// TIA Portal V18 export
// export: Created 2026-06-14T16:12:11.9430968Z, ExportSetting WithDefaults, DisplayName Totally Integrated Automation Portal, DisplayVersion V18 Update 5, DisplayName TIA Portal Openness, DisplayVersion V18 Update 5, DisplayName TIA Portal Version Control Interface, DisplayVersion V18, DisplayName SINAMICS Startdrive Advanced, DisplayVersion V18 SP2 Update 1, DisplayName SINAMICS Startdrive G110M, G120, G120C, G120D, G120P, G115D, DisplayVersion V18 SP2 Update 1, DisplayName SINAMICS Startdrive G130, G150, S120, S150, SINAMICS MV, S210, G220, S200, DisplayVersion V18 SP2 Update 1, DisplayName STEP 7 Professional, DisplayVersion V18 Update 5, DisplayName STEP 7 Safety, DisplayVersion V18, DisplayName WinCC Advanced / Unified PC, DisplayVersion V18 Update 5
FUNCTION "TEMPLATE--v1.0--06_Feedback Error" : Void   // FC7, F_LAD
TITLE = group / bypass contactor feedback errors by I/O Node
{ S7_Optimized_Access := 'TRUE' }
VERSION : 0.1
// v1.0 First Emission
// stored: AutoNumber true, IsIECCheckEnabled false, UDAEnableTagReadback false
BEGIN

REGION Network 1: !!NetworkComment$$
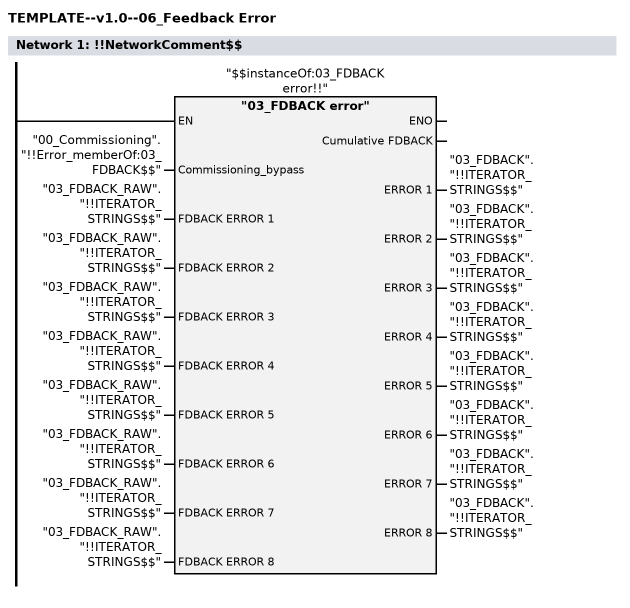
   RUNG wire#powerrail
      "$$instanceOf:03_FDBACK error!!"(Commissioning_bypass := "00_Commissioning"."!!Error_memberOf:03_FDBACK$$", "FDBACK ERROR 1" := "03_FDBACK_RAW"."!!ITERATOR_STRINGS$$", "FDBACK ERROR 2" := "03_FDBACK_RAW"."!!ITERATOR_STRINGS$$", "FDBACK ERROR 3" := "03_FDBACK_RAW"."!!ITERATOR_STRINGS$$", "FDBACK ERROR 4" := "03_FDBACK_RAW"."!!ITERATOR_STRINGS$$", "FDBACK ERROR 5" := "03_FDBACK_RAW"."!!ITERATOR_STRINGS$$", "FDBACK ERROR 6" := "03_FDBACK_RAW"."!!ITERATOR_STRINGS$$", "FDBACK ERROR 7" := "03_FDBACK_RAW"."!!ITERATOR_STRINGS$$", "FDBACK ERROR 8" := "03_FDBACK_RAW"."!!ITERATOR_STRINGS$$", "Cumulative FDBACK" =>, "ERROR 1" => "03_FDBACK"."!!ITERATOR_STRINGS$$", "ERROR 2" => "03_FDBACK"."!!ITERATOR_STRINGS$$", "ERROR 3" => "03_FDBACK"."!!ITERATOR_STRINGS$$", "ERROR 4" => "03_FDBACK"."!!ITERATOR_STRINGS$$", "ERROR 5" => "03_FDBACK"."!!ITERATOR_STRINGS$$", "ERROR 6" => "03_FDBACK"."!!ITERATOR_STRINGS$$", "ERROR 7" => "03_FDBACK"."!!ITERATOR_STRINGS$$", "ERROR 8" => "03_FDBACK"."!!ITERATOR_STRINGS$$")
   END_RUNG
   // the same network as SCL:
   "$$instanceOf:03_FDBACK error!!"(Commissioning_bypass := "00_Commissioning"."!!Error_memberOf:03_FDBACK$$",   // "03_FDBACK error"
                           "FDBACK ERROR 1" := "03_FDBACK_RAW"."!!ITERATOR_STRINGS$$",
                           "FDBACK ERROR 2" := "03_FDBACK_RAW"."!!ITERATOR_STRINGS$$",
                           "FDBACK ERROR 3" := "03_FDBACK_RAW"."!!ITERATOR_STRINGS$$",
                           "FDBACK ERROR 4" := "03_FDBACK_RAW"."!!ITERATOR_STRINGS$$",
                           "FDBACK ERROR 5" := "03_FDBACK_RAW"."!!ITERATOR_STRINGS$$",
                           "FDBACK ERROR 6" := "03_FDBACK_RAW"."!!ITERATOR_STRINGS$$",
                           "FDBACK ERROR 7" := "03_FDBACK_RAW"."!!ITERATOR_STRINGS$$",
                           "FDBACK ERROR 8" := "03_FDBACK_RAW"."!!ITERATOR_STRINGS$$",
                           "ERROR 1" => "03_FDBACK"."!!ITERATOR_STRINGS$$",
                           "ERROR 2" => "03_FDBACK"."!!ITERATOR_STRINGS$$",
                           "ERROR 3" => "03_FDBACK"."!!ITERATOR_STRINGS$$",
                           "ERROR 4" => "03_FDBACK"."!!ITERATOR_STRINGS$$",
                           "ERROR 5" => "03_FDBACK"."!!ITERATOR_STRINGS$$",
                           "ERROR 6" => "03_FDBACK"."!!ITERATOR_STRINGS$$",
                           "ERROR 7" => "03_FDBACK"."!!ITERATOR_STRINGS$$",
                           "ERROR 8" => "03_FDBACK"."!!ITERATOR_STRINGS$$");
END_REGION
END_FUNCTION
